{attribute 'qualified_only'}
{attribute 'strict'}
{attribute 'to_string'}
TYPE E_SeqNcTask :
(
	IDLE := 0,
	STOP,
	RESET,
	HOME,
	JOG,
	MOVE_ABS
);
END_TYPE

(* stored: Version 1.1.0.1, ProductVersion 3.1.4024.12
   DUT E_SeqNcTask: Id {af91c62d-b749-4f8b-b488-e5b765c287ff} *)
